// TIA Portal project "LearningFactory_4_0_24V_Task04_SortingSLD_V18" (V18)

(* hardware
DEVICE "ET 200SP-Station_1"  ET 200SP-Station
   slot 0: "Baugruppenträger_0"  Rack  6ES5 710-8MAx1
   slot 1: "PLC"  CPU 1512SP F-1 PN  6ES7 512-1SK01-0AB0  V2.8
      slot 32768: "PROFINET"  X1
   slot 2: "DO1+2"  DQ 16x24VDC/0.5A ST  6ES7 132-6BH01-0BA0  V0.0
      slot 1: "DO1+2"  DQ 16x24VDC/0.5A ST
   slot 3: "DO3+4"  DQ 16x24VDC/0.5A ST  6ES7 132-6BH01-0BA0  V0.0
      slot 1: "DO3+4"  DQ 16x24VDC/0.5A ST
   slot 4: "DO5+6"  DQ 16x24VDC/0.5A ST  6ES7 132-6BH01-0BA0  V0.0
      slot 1: "DO5+6"  DQ 16x24VDC/0.5A ST
   slot 5: "DO7-14"  DQ 4x24VDC/2A HS  6ES7 132-6BD20-0DA0  V2.0
      slot 1: "DO7-14"  DQ 4x24VDC/2A HS
   slot 6: "DO15-22"  DQ 4x24VDC/2A HS  6ES7 132-6BD20-0DA0  V2.0
      slot 1: "DO15-22"  DQ 4x24VDC/2A HS
   slot 7: "DO23-30"  DQ 4x24VDC/2A HS  6ES7 132-6BD20-0DA0  V2.0
      slot 1: "DO23-30"  DQ 4x24VDC/2A HS
   slot 8: "DI1+2"  DI 16x24VDC ST  6ES7 131-6BH01-0BA0  V0.0
      slot 1: "DI1+2"  DI 16x24VDC ST
   slot 9: "DI3+4"  DI 16x24VDC ST  6ES7 131-6BH01-0BA0  V0.0
      slot 1: "DI3+4"  DI 16x24VDC ST
   slot 10: "DI5"  DI 8x24VDC HS  6ES7 131-6BF00-0DA0  V1.0
      slot 1: "DI5"  DI 8x24VDC HS
   slot 11: "DI6"  DI 8x24VDC HS  6ES7 131-6BF00-0DA0  V1.0
      slot 1: "DI6"  DI 8x24VDC HS
   slot 12: "AI7-10"  AI 2xU ST  6ES7 134-6FB00-0BA1  V1.0
      slot 1: "AI7-10"  AI 2xU ST
   slot 13: "End"  Server module  6ES7 193-6PA00-0AA0  V1.1
      slot 1: "End"  Server module
   slot 127: "BA 2xRJ45"  BA 2xRJ45  6ES7 193-6AR00-0AA0  V0.0
      slot 32769: "Port_1"  6ES7 193-6AR00-0AA0
      slot 32770: "Port_2"  6ES7 193-6AR00-0AA0
*)

// ===== PLC "PLC"  CPU 1512SP F-1 PN =====

VAR_GLOBAL   // PLC tag table "Start_Stop"
   "IX_START" AT %I4.4 : Bool;
   "IX_STOP" AT %I4.6 : Bool;
END_VAR

VAR_GLOBAL   // PLC tag table "SLD - Sorting Line with Detection"
   "IX_SLD_PulseCounter_I1" AT %I3.0 : Bool;
   "IX_SLD_LightBarrierInlet_I2" AT %I3.1 : Bool;
   "IX_SLD_LightBarrierBehindColorSensor_I3" AT %I3.2 : Bool;
   "IW_SLD_ColorSensor_A4" AT %IW7 : Word;
   "IX_SLD_LightBarrierWhite_I5" AT %I3.3 : Bool;
   "IX_SLD_LightBarrierRed_I6" AT %I3.4 : Bool;
   "IX_SLD_LightBarrierBlue_I7" AT %I3.5 : Bool;
   "QX_SLD_M1_ConveyorBelt_Q1" AT %Q5.0 : Bool;
   "QX_SLD_Compressor_Q2" AT %Q5.1 : Bool;
   "QX_SLD_ValveFirstEjectorWhite_Q3" AT %Q5.2 : Bool;
   "QX_SLD_ValveSecondEjectorRed_Q4" AT %Q5.3 : Bool;
   "QX_SLD_ValveThirdEjectorBlue_Q5" AT %Q5.4 : Bool;
END_VAR

DATA_BLOCK "Task04_Sorting_DB"   // DB2
{ S7_Optimized_Access := 'TRUE' }
VERSION : 0.1
// stored: InstanceOfName Task04_Sorting
"Task04_Sorting"
BEGIN
END_DATA_BLOCK

FUNCTION_BLOCK "Task04_Sorting"   // FB2, SCL
{ S7_Optimized_Access := 'TRUE' }
VERSION : 0.1
   VAR_INPUT
      Start : Bool;
      Stop : Bool;
      LightBarrierInlet : Bool;
      LightBarrierBehindColorSensor : Bool;
      LightBarrierRed : Bool;
      PulseCounter : Bool;
   END_VAR
   VAR_OUTPUT
      M1_ConveyorBelt : Bool;
      ValveSecondEjectorRed : Bool;
      Compressor : Bool;
   END_VAR
   VAR
      Step_number : Int;
      R_TRIG_PulseCounter : R_TRIG;
      PositioningCounter : Int;
   END_VAR
BEGIN

   // Reset sequencer with pushbutton STOP 
   // Rücksetzen der Schrittkette  mit Taster STOP

   IF #Stop THEN
       #Step_number := 0;
   END_IF;

   // Start sequencer with pushbutton START
   // Starten der Schrittkette  mit Taster START


   CASE #Step_number OF
       0:  // Initial step / Initialschritt
           #M1_ConveyorBelt := FALSE;          // Conveyor stop / Band stoppen
           #ValveSecondEjectorRed := FALSE;    // retract Zylinder / Zylinder einfahren
           #Compressor := FALSE;               // Compressor off / Kompressor aus
           #PositioningCounter := 0;           // reset positioning counter / Zähler zum Positionieren zurücksetzen

           IF #Start  AND #LightBarrierInlet AND NOT #LightBarrierRed
           THEN
               #Step_number := #Step_number + 1;
           END_IF;

       1:  // Step 1 conveyor start / Schritt 1 Band starten
           #M1_ConveyorBelt := TRUE; // Conveyor start / Band starten

           IF #LightBarrierBehindColorSensor THEN
               #Step_number := #Step_number + 1;
           END_IF;

       2:  // Step 2 start positioning counter / Schritt 2 Zähler zum Positionieren starten
           #R_TRIG_PulseCounter(CLK:=#PulseCounter); // Positive edge detection PulseCounter / Positive Flanke an PulseCounter 
           IF #R_TRIG_PulseCounter.Q THEN
               #PositioningCounter := #PositioningCounter + 1;  // Positionieng Counter +1 / Zähler zum Positionieren +1
           END_IF;

           IF #PositioningCounter >= 8 THEN
               #Step_number := #Step_number + 1;
           END_IF;

       3:  // Step 3 conveyor stop; reset positioning counter / Schritt 3 Band stoppen; Zähler zum Positionieren zurücksetzen
           #M1_ConveyorBelt := FALSE; // Conveyor stop / Band stoppen
           #PositioningCounter := 0; // reset positioning counter / Zähler zum Positionieren zurücksetzen
           IF #PositioningCounter = 0 THEN
               #Step_number := #Step_number + 1;
           END_IF;

       4:  // Step 4 eject zylinder / Schritt 4 Zylinder ausfahren
           #ValveSecondEjectorRed := TRUE; // Eject zylinder / Zylinder ausfahren
           #Compressor := TRUE; // Compressor on / Kompressor ein

           IF #LightBarrierRed THEN
               #Step_number := #Step_number + 1;
           END_IF;

       5:  // Step 5 retract zylinder / Schritt 5 Zylinder einfahren
           #ValveSecondEjectorRed := False; // Retract zylinder / Zylinder einfahren
           #Compressor := False; // Compressor off / Kompressor aus

           IF NOT #LightBarrierRed THEN
               #Step_number := 0;
           END_IF;

       ELSE  // Statement section ELSE
           ;
   END_CASE;
END_FUNCTION_BLOCK

ORGANIZATION_BLOCK "Main"   // OB1, SCL, ProgramCycle
TITLE = "Main Program Sweep (Cycle)"
{ S7_Optimized_Access := 'TRUE' }
VERSION : 0.1
   VAR_INPUT
      Initial_Call : Bool;   // Initial call of this OB
      Remanence : Bool;   // =True, if remanent data are available
   END_VAR
BEGIN


   // Call subroutine Sorting
   // Aufruf Unterprogramm Sorting

   "Task04_Sorting_DB"(Start:="IX_START",
                       Stop:= NOT "IX_STOP",
                       LightBarrierInlet:= NOT "IX_SLD_LightBarrierInlet_I2",
                       LightBarrierBehindColorSensor:= NOT "IX_SLD_LightBarrierBehindColorSensor_I3",
                       LightBarrierRed:= NOT "IX_SLD_LightBarrierRed_I6",
                       PulseCounter:="IX_SLD_PulseCounter_I1",
                       M1_ConveyorBelt=>"QX_SLD_M1_ConveyorBelt_Q1",
                       ValveSecondEjectorRed=>"QX_SLD_ValveSecondEjectorRed_Q4",
                       Compressor=>"QX_SLD_Compressor_Q2");
END_ORGANIZATION_BLOCK